SUBAPPLICATION Uebung_006b (* RS-Flip-Flop mit 2x IE *)
  (* Standard: 61499-2 *)
  (* Version 1.0, 2023-10-23, franz *)
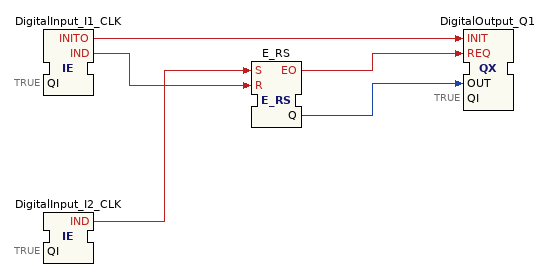
  FBS
    DigitalOutput_Q1 : QX(QI := TRUE);
    DigitalInput_I1_CLK : IE(QI := TRUE);
    DigitalInput_I2_CLK : IE(QI := TRUE);
    E_RS : E_RS;
  END_FBS
  EVENT_CONNECTIONS
    DigitalInput_I1_CLK.INITO TO DigitalOutput_Q1.INIT;
    DigitalInput_I2_CLK.IND TO E_RS.S;
    E_RS.EO TO DigitalOutput_Q1.REQ;
    DigitalInput_I1_CLK.IND TO E_RS.R;
  END_CONNECTIONS
  DATA_CONNECTIONS
    E_RS.Q TO DigitalOutput_Q1.OUT;
  END_CONNECTIONS
END_SUBAPPLICATION
